{attribute addProperty BoxType "EK1100-0000-0018"}
{attribute addProperty Id "Beckhoff_EP3xxxEK1122Beckhoff_EP3xxxEK1122_961F7095173102163.75"}
{attribute addProperty CRC "721590553"}
{attribute addProperty SizeInBites "17310"}
{attribute addProperty SizeInBytes "2163.75"}
TYPE Beckhoff_EP3xxx_2B029919 EXTENDS EK1100_179A0949 :
STRUCT
	{attribute addProperty Name "Beckhoff_EP3xxxEK1122"}
	Beckhoff_EP3xxxEK1122 : Beckhoff_EP3xxxEK1122_961F7095;
END_STRUCT
END_TYPE

(* stored: Version 1.2.0.0, ProductVersion 3.1.4024.9
   DUT Beckhoff_EP3xxx_2B029919: Id {ada232ee-4fe2-42e0-96fa-ba3b54cbbf84} *)
